FUNCTION_BLOCK FB_BasePieceHolder
VAR
    _Usable : BOOL := TRUE;
END_VAR

METHOD Equals : BOOL
VAR_INPUT
    object : ANY;
END_VAR
Equals := THIS = object.pValue;
END_METHOD

PROPERTY PUBLIC Usable : BOOL
GET
Usable := THIS^._Usable;
END_GET
SET
THIS^._Usable := Usable;
END_SET
END_PROPERTY

END_FUNCTION_BLOCK

(* stored: Version 1.1.0.1, ProductVersion 3.1.4024.12
   POU FB_BasePieceHolder: Id {a914e1f5-da13-4b28-82d8-b2b92e0b5be4}, SpecialFunc None
   Method Equals: Id {d050dfad-463d-4226-bfc9-3ebeaf2a13b0}
   Property Usable: Id {7855e544-ef20-4e89-b20f-f4776d70fc97}
   Get Get: Id {f904348c-74da-4bbd-88db-8a2063ccf759}
   Set Set: Id {35ce39aa-a1a9-4bfb-b8a8-86d265e7e6a4} *)
